PROGRAM PRG_LVCP1_Group2
VAR
    // Function Block Instance
    fbContactor: FB_ContactorControl;

    // Contactor 1 IO Structure  
    stContactor_IO: ST_ContactorIO;
    
    // Başlangıç konfigürasyonu için flag
    bContactorInitDone: BOOL := FALSE;
    bCapacitorInitDone: BOOL := FALSE;	
END_VAR



	M_Contactor();
	
	M_Capacitor();

METHOD M_Capacitor : BOOL
VAR
    nGroupIndex : INT;
END_VAR

nGroupIndex := 1;  // Grup 2 için index

IF NOT bCapacitorInitDone THEN
    // Grup 2 değerlerini ata
    GVL_LVCP1.astCompensationGroups[nGroupIndex].rPower := 25.0;
    GVL_LVCP1.astCompensationGroups[nGroupIndex].rVoltage := 450.0;
    GVL_LVCP1.astCompensationGroups[nGroupIndex].nQuantity := 8;
    GVL_LVCP1.astCompensationGroups[nGroupIndex].sTagPrefix := '+EP6-19C1';
    GVL_LVCP1.astCompensationGroups[nGroupIndex].sProductCode := 'ENT.CXD-450-25';
    
    bCapacitorInitDone := TRUE;
END_IF

// Grup 2 aktif durumu
GVL_LVCP1.abGroupActive[nGroupIndex] := stContactor_IO.bFeedback;

M_Capacitor := TRUE;
END_METHOD

METHOD M_Contactor : BOOL
VAR_INPUT
END_VAR

IF NOT bContactorInitDone THEN
    // Konfigürasyon parametreleri
    GVL_LVCP1.stGroup2_ContactorHMI.stConfig.sProjectCode := '+EP6-20K1';
    GVL_LVCP1.stGroup2_ContactorHMI.stConfig.sProductCode := 'SCH LC1G500LSEA';
    GVL_LVCP1.stGroup2_ContactorHMI.stConfig.rRatedCurrent := 500.0;
    GVL_LVCP1.stGroup2_ContactorHMI.stConfig.rRatedVoltage := 1000.0;
    GVL_LVCP1.stGroup2_ContactorHMI.stConfig.nPhaseCount := 3;
    GVL_LVCP1.stGroup2_ContactorHMI.stConfig.tFeedbackDelay := T#500MS;
    GVL_LVCP1.stGroup2_ContactorHMI.stConfig.tWeldedDelay := T#2S;
    GVL_LVCP1.stGroup2_ContactorHMI.stConfig.dwOperationLimit := 100000;
    
    // Başlangıç bakım sayacı
    GVL_LVCP1.stGroup2_ContactorHMI.stStatistics.dwRemainingOperations := GVL_LVCP1.stGroup2_ContactorHMI.stConfig.dwOperationLimit;
    
    bContactorInitDone := TRUE;
END_IF

// Function Block Çağrısı
fbContactor(
    // Fiziksel Girişler
    bFeedback := stContactor_IO.bFeedback,
    bPLCControl := stContactor_IO.bPLCControl,
    
    // Güvenlik Girişleri
    bSafetyLoop := GVL_Alarm.bSafetyLoop,
    bInterlock := FALSE,
    
    // Sistem Girişleri
    bMasterReset := GVL_Alarm.bMasterReset,
    
    // HMI Bağlantısı
    stHMI := GVL_LVCP1.stGroup2_ContactorHMI,
    
    // Fiziksel Çıkış
    bOutput => stContactor_IO.bOutput
);

M_Contactor := TRUE;
END_METHOD

END_PROGRAM

(* stored: Version 1.1.0.1, ProductVersion 3.1.4024.15
   POU PRG_LVCP1_Group2: Id {45a939ca-4d16-478f-8b9c-3b496cabdadc}, SpecialFunc None
   Method M_Capacitor: Id {d4d4cf13-b50a-4c74-a909-30e2e10b8847}
   Method M_Contactor: Id {350debfb-ab7e-479a-a823-7f73fe113b62} *)
